(* CODESYS project Library02.library
   Title: MyLibrary02
   DefaultNamespace: MyNamespace02
   Version: 1.0.0.0
   Placeholder: MyLibrary02
   Company: MyCompany

Project tree, tasks and I/O mapping:
  libraries: Tc2_Standard, * (Beckhoff Automation GmbH); Tc2_System, * (Beckhoff Automation GmbH); Tc3_Module, * (Beckhoff Automation GmbH)
  DUTs/
  GVLs/
  POUs/
    function block FB_Foo [ST]
  Version/
    global variables Global_Version
  VISUs/
*)

// Version/Global_Version
{attribute 'TcGenerated'}
// This function has been automatically generated from the project information.
VAR_GLOBAL CONSTANT
	{attribute 'const_non_replaced'}
	{attribute 'linkalways'}
	stLibVersion_MyLibrary02 : ST_LibVersion := (iMajor := 1, iMinor := 0, iBuild := 0, iRevision := 0, sVersion := '1.0.0.0');
END_VAR

// POUs/FB_Foo
FUNCTION_BLOCK PUBLIC FB_Foo
VAR_INPUT
END_VAR
VAR_OUTPUT
	{attribute 'init_namespace'}
	sNamespace	:	STRING;	
END_VAR
VAR
END_VAR

END_FUNCTION_BLOCK
